// TIA Portal V20 export
DATA_BLOCK "GLOBAL_ROBOT_DATA_DB"   // DB214
{ S7_Optimized_Access := 'TRUE' }
// stored: AutoNumber false, MemoryReserve 100
   VAR RETAIN
      Robot_HS_History_Data { ExternalWritable := 'False'} : Array[0..19] of "HS_HISTORY_EXTERNAL_UDT";
   END_VAR
BEGIN
END_DATA_BLOCK
